{attribute 'linkalways'} 
{attribute 'no_explicit_call' := 'This FB is a CLASS and must be accessed using methods or properties'}
{attribute 'enable_dynamic_creation'}
FUNCTION_BLOCK FINAL GE_USINT EXTENDS Node
VAR
	in1 : _USINT(0);
	in2 : _USINT(0);
	out : _BOOL(FALSE);
END_VAR

METHOD PUBLIC Clone : I_Node
VAR
	pNode : POINTER TO GE_USINT;
END_VAR
pNode := __NEW(GE_USINT);
Clone := pNode^;
END_METHOD

METHOD FB_init : BOOL
VAR_INPUT
	bInitRetains : BOOL; // if TRUE, the retain variables are initialized (warm start / cold start)
	bInCopyCode : BOOL;  // if TRUE, the instance afterwards gets moved into the copy code (online change)
END_VAR
AddInput('in1',THIS^.in1);
AddInput('in2',THIS^.in2);
AddOutput('out', THIS^.out);
END_METHOD

METHOD PROTECTED OnExecute
VAR
END_VAR
out.Value := in1.Value >= in2.Value;
END_METHOD

END_FUNCTION_BLOCK

(* stored: Version 1.1.0.1, ProductVersion 3.1.4024.15
   POU GE_USINT: Id {49286249-b155-4781-b367-514eee7bb3d1}, SpecialFunc None
   Folder Constructor: Id {3f29f22b-cbac-432b-a0a6-e474aa65bbf5}
   Method Clone: Id {d822936d-d0dc-4db8-b3e6-d8803775baca}
   Method FB_init: Id {7e45dfd2-4d57-4609-96bc-fe1b906067b0}
   Method OnExecute: Id {96ae001c-fd2b-4766-9b4c-8b2db10f69db} *)
